VAR_GLOBAL
	fbArbiter	:	FB_Arbiter;
	g_rTestingVelocity	:	LREAL := VISIBLE_TEST_VELOCITY;
END_VAR

VAR_GLOBAL CONSTANT
	EXCLUDED_ASSERTION_ID	:	UDINT	:= 16#FFFFFFFF; //An assertion ID that should always return "not found" in the assertion pool
	VISIBLE_TEST_VELOCITY	:	LREAL	:= 10;
	FAST_TEST_VELOCITY		:	LREAL	:= 100;
END_VAR

(* stored: Version 1.1.0.1, ProductVersion 3.1.4022.12
   GVL GVL: Id {8be29a55-f95b-0019-032e-27be63ad623d} *)
